// TIA Portal V16 export
// export: Created 2021-11-12T13:32:41.0114978Z, ExportSetting WithDefaults, DisplayName Totally Integrated Automation Portal, DisplayVersion V16 Update 3, DisplayName TIA Portal Version Control Interface, DisplayVersion V16 Update 2, DisplayName TIA Portal Openness, DisplayVersion V16 Update 3, DisplayName SINAMICS Startdrive Advanced, DisplayVersion V16 Update 5, DisplayName SINAMICS Startdrive G130, G150, S120, S150, SINAMICS MV, S210, DisplayVersion V16 Update 5, DisplayName SINAMICS Startdrive G110M, G120, G120C, G120D, G120P, G115D, DisplayVersion V16 Update 5, DisplayName STEP 7 Professional, DisplayVersion V16 Update 3, DisplayName STEP 7 Safety, DisplayVersion V16, DisplayName WinCC UA Professional, DisplayVersion V16 Update 3
FUNCTION_BLOCK "IM_200+UH11-KF10"   // FB26, LAD
TITLE = Inputs reading
{ S7_Optimized_Access := 'TRUE' }
VERSION : 0.1
// MICE Wood interface block
// stored: AutoNumber true, IsIECCheckEnabled false, IsRetainMemResEnabled false, MemoryReserve 100, SetENOAutomatically false, UDAEnableTagReadback false
   VAR
      KF11_Ix0 { S7_SetPoint := 'True'} : "STD_CH_DI";
      KF11_Ix1 { S7_SetPoint := 'True'} : "STD_CH_DI";
      KF11_Ix2 { S7_SetPoint := 'True'} : "STD_CH_DI";
      KF11_Ix3 { S7_SetPoint := 'True'} : "STD_CH_DI";
      KF11_Ix4 { S7_SetPoint := 'True'} : "STD_CH_DI";
      KF11_Ix5 { S7_SetPoint := 'True'} : "STD_CH_DI";
      KF11_Ix6 { S7_SetPoint := 'True'} : "STD_CH_DI";
      KF11_Ix7 { S7_SetPoint := 'True'} : "STD_CH_DI";
      KF11_Ix8 { S7_SetPoint := 'True'} : "STD_CH_DI";
      KF11_Ix9 { S7_SetPoint := 'True'} : "STD_CH_DI";
      KF11_Ix10 { S7_SetPoint := 'True'} : "STD_CH_DI";
      KF11_Ix11 { S7_SetPoint := 'True'} : "STD_CH_DI";
      KF11_Ix12 { S7_SetPoint := 'True'} : "STD_CH_DI";
      KF11_Ix13 { S7_SetPoint := 'True'} : "STD_CH_DI";
      KF11_Ix14 { S7_SetPoint := 'True'} : "STD_CH_DI";
      KF11_Ix15 { S7_SetPoint := 'True'} : "STD_CH_DI";
      KF12_Ix0 { S7_SetPoint := 'True'} : "STD_CH_DI";
      KF12_Ix1 { S7_SetPoint := 'True'} : "STD_CH_DI";
      KF12_Ix2 { S7_SetPoint := 'True'} : "STD_CH_DI";
      KF12_Ix3 { S7_SetPoint := 'True'} : "STD_CH_DI";
      KF12_Ix4 { S7_SetPoint := 'True'} : "STD_CH_DI";
      KF12_Ix5 { S7_SetPoint := 'True'} : "STD_CH_DI";
      KF12_Ix6 { S7_SetPoint := 'True'} : "STD_CH_DI";
      KF12_Ix7 { S7_SetPoint := 'True'} : "STD_CH_DI";
      KF12_Ix8 { S7_SetPoint := 'True'} : "STD_CH_DI";
      KF12_Ix9 { S7_SetPoint := 'True'} : "STD_CH_DI";
      KF12_Ix10 { S7_SetPoint := 'True'} : "STD_CH_DI";
      KF12_Ix11 { S7_SetPoint := 'True'} : "STD_CH_DI";
      KF12_Ix12 { S7_SetPoint := 'True'} : "STD_CH_DI";
      KF12_Ix13 { S7_SetPoint := 'True'} : "STD_CH_DI";
      KF12_Ix14 { S7_SetPoint := 'True'} : "STD_CH_DI";
      KF12_Ix15 { S7_SetPoint := 'True'} : "STD_CH_DI";
      KF13_Ix0 { S7_SetPoint := 'True'} : "STD_CH_DI";
      KF13_Ix1 { S7_SetPoint := 'True'} : "STD_CH_DI";
      KF13_Ix2 { S7_SetPoint := 'True'} : "STD_CH_DI";
      KF13_Ix3 { S7_SetPoint := 'True'} : "STD_CH_DI";
      KF13_Ix4 { S7_SetPoint := 'True'} : "STD_CH_DI";
      KF13_Ix5 { S7_SetPoint := 'True'} : "STD_CH_DI";
      KF13_Ix6 { S7_SetPoint := 'True'} : "STD_CH_DI";
      KF13_Ix7 { S7_SetPoint := 'True'} : "STD_CH_DI";
      KF13_Ix8 { S7_SetPoint := 'True'} : "STD_CH_DI";
      KF13_Ix9 { S7_SetPoint := 'True'} : "STD_CH_DI";
      KF13_Ix10 { S7_SetPoint := 'True'} : "STD_CH_DI";
      KF13_Ix11 { S7_SetPoint := 'True'} : "STD_CH_DI";
      KF13_Ix12 { S7_SetPoint := 'True'} : "STD_CH_DI";
      KF13_Ix13 { S7_SetPoint := 'True'} : "STD_CH_DI";
      KF13_Ix14 { S7_SetPoint := 'True'} : "STD_CH_DI";
      KF13_Ix15 { S7_SetPoint := 'True'} : "STD_CH_DI";
      KF14_Ix0 { S7_SetPoint := 'True'} : "STD_CH_DI";
      KF14_Ix1 { S7_SetPoint := 'True'} : "STD_CH_DI";
      KF14_Ix2 { S7_SetPoint := 'True'} : "STD_CH_DI";
      KF14_Ix3 { S7_SetPoint := 'True'} : "STD_CH_DI";
      KF14_Ix4 { S7_SetPoint := 'True'} : "STD_CH_DI";
      KF14_Ix5 { S7_SetPoint := 'True'} : "STD_CH_DI";
      KF14_Ix6 { S7_SetPoint := 'True'} : "STD_CH_DI";
      KF14_Ix7 { S7_SetPoint := 'True'} : "STD_CH_DI";
      KF14_Ix8 { S7_SetPoint := 'True'} : "STD_CH_DI";
      KF14_Ix9 { S7_SetPoint := 'True'} : "STD_CH_DI";
      KF14_Ix10 { S7_SetPoint := 'True'} : "STD_CH_DI";
      KF14_Ix11 { S7_SetPoint := 'True'} : "STD_CH_DI";
      KF14_Ix12 { S7_SetPoint := 'True'} : "STD_CH_DI";
      KF14_Ix13 { S7_SetPoint := 'True'} : "STD_CH_DI";
      KF14_Ix14 { S7_SetPoint := 'True'} : "STD_CH_DI";
      KF14_Ix15 { S7_SetPoint := 'True'} : "STD_CH_DI";
      KF15_Ix0 { S7_SetPoint := 'True'} : "STD_CH_DI";
      KF15_Ix1 { S7_SetPoint := 'True'} : "STD_CH_DI";
      KF15_Ix2 { S7_SetPoint := 'True'} : "STD_CH_DI";
      KF15_Ix3 { S7_SetPoint := 'True'} : "STD_CH_DI";
      KF15_Ix4 { S7_SetPoint := 'True'} : "STD_CH_DI";
      KF15_Ix5 { S7_SetPoint := 'True'} : "STD_CH_DI";
      KF15_Ix6 { S7_SetPoint := 'True'} : "STD_CH_DI";
      KF15_Ix7 { S7_SetPoint := 'True'} : "STD_CH_DI";
      KF61_AI0 { S7_SetPoint := 'True'} : "STD_CH_AI";
      KF61_AI1 { S7_SetPoint := 'True'} : "STD_CH_AI";
      KF61_AI2 { S7_SetPoint := 'True'} : "STD_CH_AI";
      KF61_AI3 { S7_SetPoint := 'True'} : "STD_CH_AI";
   END_VAR
   VAR_TEMP   // added for the SCL form of the ladder/FBD networks
      _w1 : Bool;
      _w2 : Bool;
      _w3 : Bool;
      _w4 : Bool;
      _w5 : Bool;
      _w6 : Bool;
      _w7 : Bool;
      _w8 : Bool;
   END_VAR
BEGIN

REGION Network 1: Module position -KF11
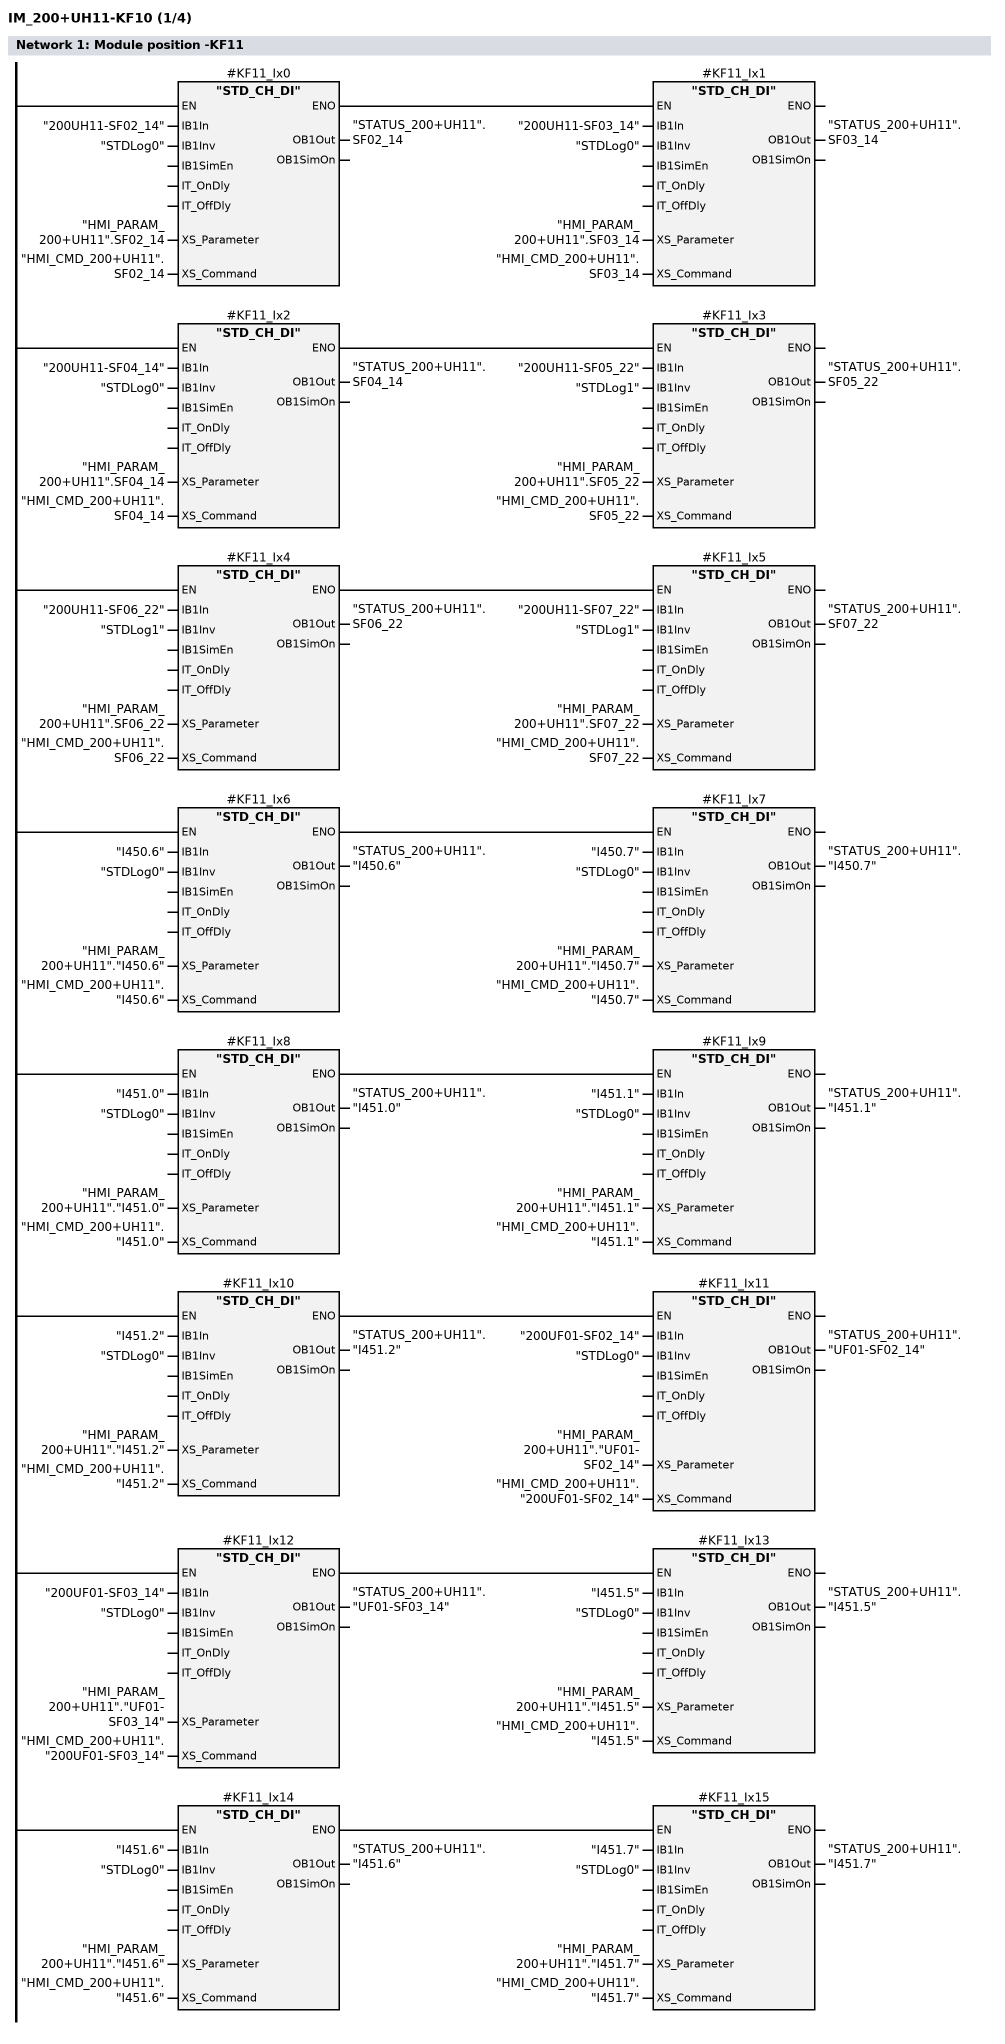
   RUNG wire#powerrail
      #KF11_Ix0(IB1In := "200UH11-SF02_14", IB1Inv := "STDLog0", IB1SimEn :=, IT_OnDly :=, IT_OffDly :=, XS_Parameter := "HMI_PARAM_200+UH11".SF02_14, XS_Command := "HMI_CMD_200+UH11".SF02_14, OB1Out => "STATUS_200+UH11".SF02_14, OB1SimOn =>)
      #KF11_Ix1(IB1In := "200UH11-SF03_14", IB1Inv := "STDLog0", IB1SimEn :=, IT_OnDly :=, IT_OffDly :=, XS_Parameter := "HMI_PARAM_200+UH11".SF03_14, XS_Command := "HMI_CMD_200+UH11".SF03_14, OB1Out => "STATUS_200+UH11".SF03_14, OB1SimOn =>)
   END_RUNG
   RUNG wire#powerrail
      #KF11_Ix2(IB1In := "200UH11-SF04_14", IB1Inv := "STDLog0", IB1SimEn :=, IT_OnDly :=, IT_OffDly :=, XS_Parameter := "HMI_PARAM_200+UH11".SF04_14, XS_Command := "HMI_CMD_200+UH11".SF04_14, OB1Out => "STATUS_200+UH11".SF04_14, OB1SimOn =>)
      #KF11_Ix3(IB1In := "200UH11-SF05_22", IB1Inv := "STDLog1", IB1SimEn :=, IT_OnDly :=, IT_OffDly :=, XS_Parameter := "HMI_PARAM_200+UH11".SF05_22, XS_Command := "HMI_CMD_200+UH11".SF05_22, OB1Out => "STATUS_200+UH11".SF05_22, OB1SimOn =>)
   END_RUNG
   RUNG wire#powerrail
      #KF11_Ix4(IB1In := "200UH11-SF06_22", IB1Inv := "STDLog1", IB1SimEn :=, IT_OnDly :=, IT_OffDly :=, XS_Parameter := "HMI_PARAM_200+UH11".SF06_22, XS_Command := "HMI_CMD_200+UH11".SF06_22, OB1Out => "STATUS_200+UH11".SF06_22, OB1SimOn =>)
      #KF11_Ix5(IB1In := "200UH11-SF07_22", IB1Inv := "STDLog1", IB1SimEn :=, IT_OnDly :=, IT_OffDly :=, XS_Parameter := "HMI_PARAM_200+UH11".SF07_22, XS_Command := "HMI_CMD_200+UH11".SF07_22, OB1Out => "STATUS_200+UH11".SF07_22, OB1SimOn =>)
   END_RUNG
   RUNG wire#powerrail
      #KF11_Ix6(IB1In := "I450.6", IB1Inv := "STDLog0", IB1SimEn :=, IT_OnDly :=, IT_OffDly :=, XS_Parameter := "HMI_PARAM_200+UH11"."I450.6", XS_Command := "HMI_CMD_200+UH11"."I450.6", OB1Out => "STATUS_200+UH11"."I450.6", OB1SimOn =>)
      #KF11_Ix7(IB1In := "I450.7", IB1Inv := "STDLog0", IB1SimEn :=, IT_OnDly :=, IT_OffDly :=, XS_Parameter := "HMI_PARAM_200+UH11"."I450.7", XS_Command := "HMI_CMD_200+UH11"."I450.7", OB1Out => "STATUS_200+UH11"."I450.7", OB1SimOn =>)
   END_RUNG
   RUNG wire#powerrail
      #KF11_Ix8(IB1In := "I451.0", IB1Inv := "STDLog0", IB1SimEn :=, IT_OnDly :=, IT_OffDly :=, XS_Parameter := "HMI_PARAM_200+UH11"."I451.0", XS_Command := "HMI_CMD_200+UH11"."I451.0", OB1Out => "STATUS_200+UH11"."I451.0", OB1SimOn =>)
      #KF11_Ix9(IB1In := "I451.1", IB1Inv := "STDLog0", IB1SimEn :=, IT_OnDly :=, IT_OffDly :=, XS_Parameter := "HMI_PARAM_200+UH11"."I451.1", XS_Command := "HMI_CMD_200+UH11"."I451.1", OB1Out => "STATUS_200+UH11"."I451.1", OB1SimOn =>)
   END_RUNG
   RUNG wire#powerrail
      #KF11_Ix10(IB1In := "I451.2", IB1Inv := "STDLog0", IB1SimEn :=, IT_OnDly :=, IT_OffDly :=, XS_Parameter := "HMI_PARAM_200+UH11"."I451.2", XS_Command := "HMI_CMD_200+UH11"."I451.2", OB1Out => "STATUS_200+UH11"."I451.2", OB1SimOn =>)
      #KF11_Ix11(IB1In := "200UF01-SF02_14", IB1Inv := "STDLog0", IB1SimEn :=, IT_OnDly :=, IT_OffDly :=, XS_Parameter := "HMI_PARAM_200+UH11"."UF01-SF02_14", XS_Command := "HMI_CMD_200+UH11"."200UF01-SF02_14", OB1Out => "STATUS_200+UH11"."UF01-SF02_14", OB1SimOn =>)
   END_RUNG
   RUNG wire#powerrail
      #KF11_Ix12(IB1In := "200UF01-SF03_14", IB1Inv := "STDLog0", IB1SimEn :=, IT_OnDly :=, IT_OffDly :=, XS_Parameter := "HMI_PARAM_200+UH11"."UF01-SF03_14", XS_Command := "HMI_CMD_200+UH11"."200UF01-SF03_14", OB1Out => "STATUS_200+UH11"."UF01-SF03_14", OB1SimOn =>)
      #KF11_Ix13(IB1In := "I451.5", IB1Inv := "STDLog0", IB1SimEn :=, IT_OnDly :=, IT_OffDly :=, XS_Parameter := "HMI_PARAM_200+UH11"."I451.5", XS_Command := "HMI_CMD_200+UH11"."I451.5", OB1Out => "STATUS_200+UH11"."I451.5", OB1SimOn =>)
   END_RUNG
   RUNG wire#powerrail
      #KF11_Ix14(IB1In := "I451.6", IB1Inv := "STDLog0", IB1SimEn :=, IT_OnDly :=, IT_OffDly :=, XS_Parameter := "HMI_PARAM_200+UH11"."I451.6", XS_Command := "HMI_CMD_200+UH11"."I451.6", OB1Out => "STATUS_200+UH11"."I451.6", OB1SimOn =>)
      #KF11_Ix15(IB1In := "I451.7", IB1Inv := "STDLog0", IB1SimEn :=, IT_OnDly :=, IT_OffDly :=, XS_Parameter := "HMI_PARAM_200+UH11"."I451.7", XS_Command := "HMI_CMD_200+UH11"."I451.7", OB1Out => "STATUS_200+UH11"."I451.7", OB1SimOn =>)
   END_RUNG
   // the same network as SCL:
   #KF11_Ix0(IB1In := "200UH11-SF02_14",   // "STD_CH_DI"
             IB1Inv := "STDLog0",
             XS_Parameter := "HMI_PARAM_200+UH11".SF02_14,
             XS_Command := "HMI_CMD_200+UH11".SF02_14,
             OB1Out => "STATUS_200+UH11".SF02_14,
             ENO => #_w1);
   IF #_w1 THEN
       #KF11_Ix1(IB1In := "200UH11-SF03_14",   // "STD_CH_DI"
                 IB1Inv := "STDLog0",
                 XS_Parameter := "HMI_PARAM_200+UH11".SF03_14,
                 XS_Command := "HMI_CMD_200+UH11".SF03_14,
                 OB1Out => "STATUS_200+UH11".SF03_14);
   END_IF;
   #KF11_Ix2(IB1In := "200UH11-SF04_14",   // "STD_CH_DI"
             IB1Inv := "STDLog0",
             XS_Parameter := "HMI_PARAM_200+UH11".SF04_14,
             XS_Command := "HMI_CMD_200+UH11".SF04_14,
             OB1Out => "STATUS_200+UH11".SF04_14,
             ENO => #_w2);
   IF #_w2 THEN
       #KF11_Ix3(IB1In := "200UH11-SF05_22",   // "STD_CH_DI"
                 IB1Inv := "STDLog1",
                 XS_Parameter := "HMI_PARAM_200+UH11".SF05_22,
                 XS_Command := "HMI_CMD_200+UH11".SF05_22,
                 OB1Out => "STATUS_200+UH11".SF05_22);
   END_IF;
   #KF11_Ix4(IB1In := "200UH11-SF06_22",   // "STD_CH_DI"
             IB1Inv := "STDLog1",
             XS_Parameter := "HMI_PARAM_200+UH11".SF06_22,
             XS_Command := "HMI_CMD_200+UH11".SF06_22,
             OB1Out => "STATUS_200+UH11".SF06_22,
             ENO => #_w3);
   IF #_w3 THEN
       #KF11_Ix5(IB1In := "200UH11-SF07_22",   // "STD_CH_DI"
                 IB1Inv := "STDLog1",
                 XS_Parameter := "HMI_PARAM_200+UH11".SF07_22,
                 XS_Command := "HMI_CMD_200+UH11".SF07_22,
                 OB1Out => "STATUS_200+UH11".SF07_22);
   END_IF;
   #KF11_Ix6(IB1In := "I450.6",   // "STD_CH_DI"
             IB1Inv := "STDLog0",
             XS_Parameter := "HMI_PARAM_200+UH11"."I450.6",
             XS_Command := "HMI_CMD_200+UH11"."I450.6",
             OB1Out => "STATUS_200+UH11"."I450.6",
             ENO => #_w4);
   IF #_w4 THEN
       #KF11_Ix7(IB1In := "I450.7",   // "STD_CH_DI"
                 IB1Inv := "STDLog0",
                 XS_Parameter := "HMI_PARAM_200+UH11"."I450.7",
                 XS_Command := "HMI_CMD_200+UH11"."I450.7",
                 OB1Out => "STATUS_200+UH11"."I450.7");
   END_IF;
   #KF11_Ix8(IB1In := "I451.0",   // "STD_CH_DI"
             IB1Inv := "STDLog0",
             XS_Parameter := "HMI_PARAM_200+UH11"."I451.0",
             XS_Command := "HMI_CMD_200+UH11"."I451.0",
             OB1Out => "STATUS_200+UH11"."I451.0",
             ENO => #_w5);
   IF #_w5 THEN
       #KF11_Ix9(IB1In := "I451.1",   // "STD_CH_DI"
                 IB1Inv := "STDLog0",
                 XS_Parameter := "HMI_PARAM_200+UH11"."I451.1",
                 XS_Command := "HMI_CMD_200+UH11"."I451.1",
                 OB1Out => "STATUS_200+UH11"."I451.1");
   END_IF;
   #KF11_Ix10(IB1In := "I451.2",   // "STD_CH_DI"
              IB1Inv := "STDLog0",
              XS_Parameter := "HMI_PARAM_200+UH11"."I451.2",
              XS_Command := "HMI_CMD_200+UH11"."I451.2",
              OB1Out => "STATUS_200+UH11"."I451.2",
              ENO => #_w6);
   IF #_w6 THEN
       #KF11_Ix11(IB1In := "200UF01-SF02_14",   // "STD_CH_DI"
                  IB1Inv := "STDLog0",
                  XS_Parameter := "HMI_PARAM_200+UH11"."UF01-SF02_14",
                  XS_Command := "HMI_CMD_200+UH11"."200UF01-SF02_14",
                  OB1Out => "STATUS_200+UH11"."UF01-SF02_14");
   END_IF;
   #KF11_Ix12(IB1In := "200UF01-SF03_14",   // "STD_CH_DI"
              IB1Inv := "STDLog0",
              XS_Parameter := "HMI_PARAM_200+UH11"."UF01-SF03_14",
              XS_Command := "HMI_CMD_200+UH11"."200UF01-SF03_14",
              OB1Out => "STATUS_200+UH11"."UF01-SF03_14",
              ENO => #_w7);
   IF #_w7 THEN
       #KF11_Ix13(IB1In := "I451.5",   // "STD_CH_DI"
                  IB1Inv := "STDLog0",
                  XS_Parameter := "HMI_PARAM_200+UH11"."I451.5",
                  XS_Command := "HMI_CMD_200+UH11"."I451.5",
                  OB1Out => "STATUS_200+UH11"."I451.5");
   END_IF;
   #KF11_Ix14(IB1In := "I451.6",   // "STD_CH_DI"
              IB1Inv := "STDLog0",
              XS_Parameter := "HMI_PARAM_200+UH11"."I451.6",
              XS_Command := "HMI_CMD_200+UH11"."I451.6",
              OB1Out => "STATUS_200+UH11"."I451.6",
              ENO => #_w8);
   IF #_w8 THEN
       #KF11_Ix15(IB1In := "I451.7",   // "STD_CH_DI"
                  IB1Inv := "STDLog0",
                  XS_Parameter := "HMI_PARAM_200+UH11"."I451.7",
                  XS_Command := "HMI_CMD_200+UH11"."I451.7",
                  OB1Out => "STATUS_200+UH11"."I451.7");
   END_IF;
END_REGION

REGION Network 2: Module position -KF12
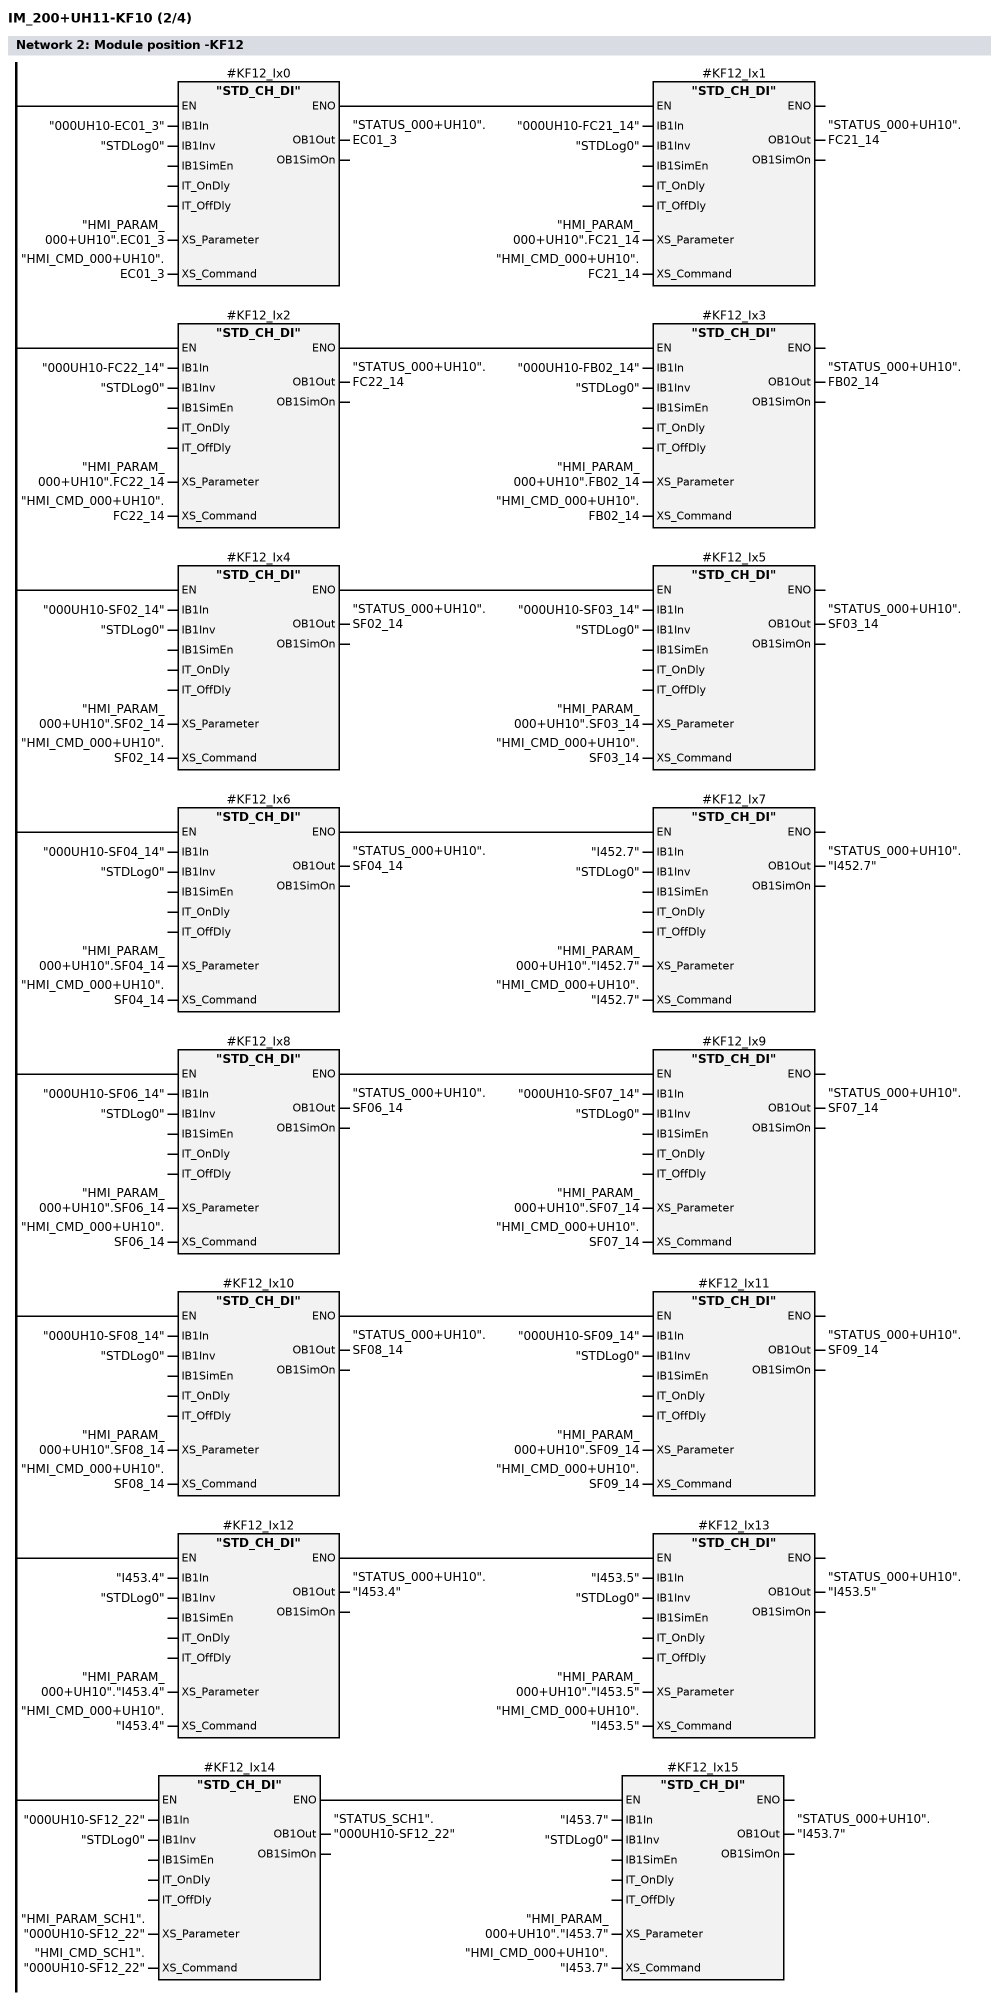
   RUNG wire#powerrail
      #KF12_Ix0(IB1In := "000UH10-EC01_3", IB1Inv := "STDLog0", IB1SimEn :=, IT_OnDly :=, IT_OffDly :=, XS_Parameter := "HMI_PARAM_000+UH10".EC01_3, XS_Command := "HMI_CMD_000+UH10".EC01_3, OB1Out => "STATUS_000+UH10".EC01_3, OB1SimOn =>)
      #KF12_Ix1(IB1In := "000UH10-FC21_14", IB1Inv := "STDLog0", IB1SimEn :=, IT_OnDly :=, IT_OffDly :=, XS_Parameter := "HMI_PARAM_000+UH10".FC21_14, XS_Command := "HMI_CMD_000+UH10".FC21_14, OB1Out => "STATUS_000+UH10".FC21_14, OB1SimOn =>)
   END_RUNG
   RUNG wire#powerrail
      #KF12_Ix2(IB1In := "000UH10-FC22_14", IB1Inv := "STDLog0", IB1SimEn :=, IT_OnDly :=, IT_OffDly :=, XS_Parameter := "HMI_PARAM_000+UH10".FC22_14, XS_Command := "HMI_CMD_000+UH10".FC22_14, OB1Out => "STATUS_000+UH10".FC22_14, OB1SimOn =>)
      #KF12_Ix3(IB1In := "000UH10-FB02_14", IB1Inv := "STDLog0", IB1SimEn :=, IT_OnDly :=, IT_OffDly :=, XS_Parameter := "HMI_PARAM_000+UH10".FB02_14, XS_Command := "HMI_CMD_000+UH10".FB02_14, OB1Out => "STATUS_000+UH10".FB02_14, OB1SimOn =>)
   END_RUNG
   RUNG wire#powerrail
      #KF12_Ix4(IB1In := "000UH10-SF02_14", IB1Inv := "STDLog0", IB1SimEn :=, IT_OnDly :=, IT_OffDly :=, XS_Parameter := "HMI_PARAM_000+UH10".SF02_14, XS_Command := "HMI_CMD_000+UH10".SF02_14, OB1Out => "STATUS_000+UH10".SF02_14, OB1SimOn =>)
      #KF12_Ix5(IB1In := "000UH10-SF03_14", IB1Inv := "STDLog0", IB1SimEn :=, IT_OnDly :=, IT_OffDly :=, XS_Parameter := "HMI_PARAM_000+UH10".SF03_14, XS_Command := "HMI_CMD_000+UH10".SF03_14, OB1Out => "STATUS_000+UH10".SF03_14, OB1SimOn =>)
   END_RUNG
   RUNG wire#powerrail
      #KF12_Ix6(IB1In := "000UH10-SF04_14", IB1Inv := "STDLog0", IB1SimEn :=, IT_OnDly :=, IT_OffDly :=, XS_Parameter := "HMI_PARAM_000+UH10".SF04_14, XS_Command := "HMI_CMD_000+UH10".SF04_14, OB1Out => "STATUS_000+UH10".SF04_14, OB1SimOn =>)
      #KF12_Ix7(IB1In := "I452.7", IB1Inv := "STDLog0", IB1SimEn :=, IT_OnDly :=, IT_OffDly :=, XS_Parameter := "HMI_PARAM_000+UH10"."I452.7", XS_Command := "HMI_CMD_000+UH10"."I452.7", OB1Out => "STATUS_000+UH10"."I452.7", OB1SimOn =>)
   END_RUNG
   RUNG wire#powerrail
      #KF12_Ix8(IB1In := "000UH10-SF06_14", IB1Inv := "STDLog0", IB1SimEn :=, IT_OnDly :=, IT_OffDly :=, XS_Parameter := "HMI_PARAM_000+UH10".SF06_14, XS_Command := "HMI_CMD_000+UH10".SF06_14, OB1Out => "STATUS_000+UH10".SF06_14, OB1SimOn =>)
      #KF12_Ix9(IB1In := "000UH10-SF07_14", IB1Inv := "STDLog0", IB1SimEn :=, IT_OnDly :=, IT_OffDly :=, XS_Parameter := "HMI_PARAM_000+UH10".SF07_14, XS_Command := "HMI_CMD_000+UH10".SF07_14, OB1Out => "STATUS_000+UH10".SF07_14, OB1SimOn =>)
   END_RUNG
   RUNG wire#powerrail
      #KF12_Ix10(IB1In := "000UH10-SF08_14", IB1Inv := "STDLog0", IB1SimEn :=, IT_OnDly :=, IT_OffDly :=, XS_Parameter := "HMI_PARAM_000+UH10".SF08_14, XS_Command := "HMI_CMD_000+UH10".SF08_14, OB1Out => "STATUS_000+UH10".SF08_14, OB1SimOn =>)
      #KF12_Ix11(IB1In := "000UH10-SF09_14", IB1Inv := "STDLog0", IB1SimEn :=, IT_OnDly :=, IT_OffDly :=, XS_Parameter := "HMI_PARAM_000+UH10".SF09_14, XS_Command := "HMI_CMD_000+UH10".SF09_14, OB1Out => "STATUS_000+UH10".SF09_14, OB1SimOn =>)
   END_RUNG
   RUNG wire#powerrail
      #KF12_Ix12(IB1In := "I453.4", IB1Inv := "STDLog0", IB1SimEn :=, IT_OnDly :=, IT_OffDly :=, XS_Parameter := "HMI_PARAM_000+UH10"."I453.4", XS_Command := "HMI_CMD_000+UH10"."I453.4", OB1Out => "STATUS_000+UH10"."I453.4", OB1SimOn =>)
      #KF12_Ix13(IB1In := "I453.5", IB1Inv := "STDLog0", IB1SimEn :=, IT_OnDly :=, IT_OffDly :=, XS_Parameter := "HMI_PARAM_000+UH10"."I453.5", XS_Command := "HMI_CMD_000+UH10"."I453.5", OB1Out => "STATUS_000+UH10"."I453.5", OB1SimOn =>)
   END_RUNG
   RUNG wire#powerrail
      #KF12_Ix14(IB1In := "000UH10-SF12_22", IB1Inv := "STDLog0", IB1SimEn :=, IT_OnDly :=, IT_OffDly :=, XS_Parameter := "HMI_PARAM_SCH1"."000UH10-SF12_22", XS_Command := "HMI_CMD_SCH1"."000UH10-SF12_22", OB1Out => "STATUS_SCH1"."000UH10-SF12_22", OB1SimOn =>)
      #KF12_Ix15(IB1In := "I453.7", IB1Inv := "STDLog0", IB1SimEn :=, IT_OnDly :=, IT_OffDly :=, XS_Parameter := "HMI_PARAM_000+UH10"."I453.7", XS_Command := "HMI_CMD_000+UH10"."I453.7", OB1Out => "STATUS_000+UH10"."I453.7", OB1SimOn =>)
   END_RUNG
   // the same network as SCL:
   #KF12_Ix0(IB1In := "000UH10-EC01_3",   // "STD_CH_DI"
             IB1Inv := "STDLog0",
             XS_Parameter := "HMI_PARAM_000+UH10".EC01_3,
             XS_Command := "HMI_CMD_000+UH10".EC01_3,
             OB1Out => "STATUS_000+UH10".EC01_3,
             ENO => #_w1);
   IF #_w1 THEN
       #KF12_Ix1(IB1In := "000UH10-FC21_14",   // "STD_CH_DI"
                 IB1Inv := "STDLog0",
                 XS_Parameter := "HMI_PARAM_000+UH10".FC21_14,
                 XS_Command := "HMI_CMD_000+UH10".FC21_14,
                 OB1Out => "STATUS_000+UH10".FC21_14);
   END_IF;
   #KF12_Ix2(IB1In := "000UH10-FC22_14",   // "STD_CH_DI"
             IB1Inv := "STDLog0",
             XS_Parameter := "HMI_PARAM_000+UH10".FC22_14,
             XS_Command := "HMI_CMD_000+UH10".FC22_14,
             OB1Out => "STATUS_000+UH10".FC22_14,
             ENO => #_w2);
   IF #_w2 THEN
       #KF12_Ix3(IB1In := "000UH10-FB02_14",   // "STD_CH_DI"
                 IB1Inv := "STDLog0",
                 XS_Parameter := "HMI_PARAM_000+UH10".FB02_14,
                 XS_Command := "HMI_CMD_000+UH10".FB02_14,
                 OB1Out => "STATUS_000+UH10".FB02_14);
   END_IF;
   #KF12_Ix4(IB1In := "000UH10-SF02_14",   // "STD_CH_DI"
             IB1Inv := "STDLog0",
             XS_Parameter := "HMI_PARAM_000+UH10".SF02_14,
             XS_Command := "HMI_CMD_000+UH10".SF02_14,
             OB1Out => "STATUS_000+UH10".SF02_14,
             ENO => #_w3);
   IF #_w3 THEN
       #KF12_Ix5(IB1In := "000UH10-SF03_14",   // "STD_CH_DI"
                 IB1Inv := "STDLog0",
                 XS_Parameter := "HMI_PARAM_000+UH10".SF03_14,
                 XS_Command := "HMI_CMD_000+UH10".SF03_14,
                 OB1Out => "STATUS_000+UH10".SF03_14);
   END_IF;
   #KF12_Ix6(IB1In := "000UH10-SF04_14",   // "STD_CH_DI"
             IB1Inv := "STDLog0",
             XS_Parameter := "HMI_PARAM_000+UH10".SF04_14,
             XS_Command := "HMI_CMD_000+UH10".SF04_14,
             OB1Out => "STATUS_000+UH10".SF04_14,
             ENO => #_w4);
   IF #_w4 THEN
       #KF12_Ix7(IB1In := "I452.7",   // "STD_CH_DI"
                 IB1Inv := "STDLog0",
                 XS_Parameter := "HMI_PARAM_000+UH10"."I452.7",
                 XS_Command := "HMI_CMD_000+UH10"."I452.7",
                 OB1Out => "STATUS_000+UH10"."I452.7");
   END_IF;
   #KF12_Ix8(IB1In := "000UH10-SF06_14",   // "STD_CH_DI"
             IB1Inv := "STDLog0",
             XS_Parameter := "HMI_PARAM_000+UH10".SF06_14,
             XS_Command := "HMI_CMD_000+UH10".SF06_14,
             OB1Out => "STATUS_000+UH10".SF06_14,
             ENO => #_w5);
   IF #_w5 THEN
       #KF12_Ix9(IB1In := "000UH10-SF07_14",   // "STD_CH_DI"
                 IB1Inv := "STDLog0",
                 XS_Parameter := "HMI_PARAM_000+UH10".SF07_14,
                 XS_Command := "HMI_CMD_000+UH10".SF07_14,
                 OB1Out => "STATUS_000+UH10".SF07_14);
   END_IF;
   #KF12_Ix10(IB1In := "000UH10-SF08_14",   // "STD_CH_DI"
              IB1Inv := "STDLog0",
              XS_Parameter := "HMI_PARAM_000+UH10".SF08_14,
              XS_Command := "HMI_CMD_000+UH10".SF08_14,
              OB1Out => "STATUS_000+UH10".SF08_14,
              ENO => #_w6);
   IF #_w6 THEN
       #KF12_Ix11(IB1In := "000UH10-SF09_14",   // "STD_CH_DI"
                  IB1Inv := "STDLog0",
                  XS_Parameter := "HMI_PARAM_000+UH10".SF09_14,
                  XS_Command := "HMI_CMD_000+UH10".SF09_14,
                  OB1Out => "STATUS_000+UH10".SF09_14);
   END_IF;
   #KF12_Ix12(IB1In := "I453.4",   // "STD_CH_DI"
              IB1Inv := "STDLog0",
              XS_Parameter := "HMI_PARAM_000+UH10"."I453.4",
              XS_Command := "HMI_CMD_000+UH10"."I453.4",
              OB1Out => "STATUS_000+UH10"."I453.4",
              ENO => #_w7);
   IF #_w7 THEN
       #KF12_Ix13(IB1In := "I453.5",   // "STD_CH_DI"
                  IB1Inv := "STDLog0",
                  XS_Parameter := "HMI_PARAM_000+UH10"."I453.5",
                  XS_Command := "HMI_CMD_000+UH10"."I453.5",
                  OB1Out => "STATUS_000+UH10"."I453.5");
   END_IF;
   #KF12_Ix14(IB1In := "000UH10-SF12_22",   // "STD_CH_DI"
              IB1Inv := "STDLog0",
              XS_Parameter := "HMI_PARAM_SCH1"."000UH10-SF12_22",
              XS_Command := "HMI_CMD_SCH1"."000UH10-SF12_22",
              OB1Out => "STATUS_SCH1"."000UH10-SF12_22",
              ENO => #_w8);
   IF #_w8 THEN
       #KF12_Ix15(IB1In := "I453.7",   // "STD_CH_DI"
                  IB1Inv := "STDLog0",
                  XS_Parameter := "HMI_PARAM_000+UH10"."I453.7",
                  XS_Command := "HMI_CMD_000+UH10"."I453.7",
                  OB1Out => "STATUS_000+UH10"."I453.7");
   END_IF;
END_REGION

REGION Network 3: Module position -KF13
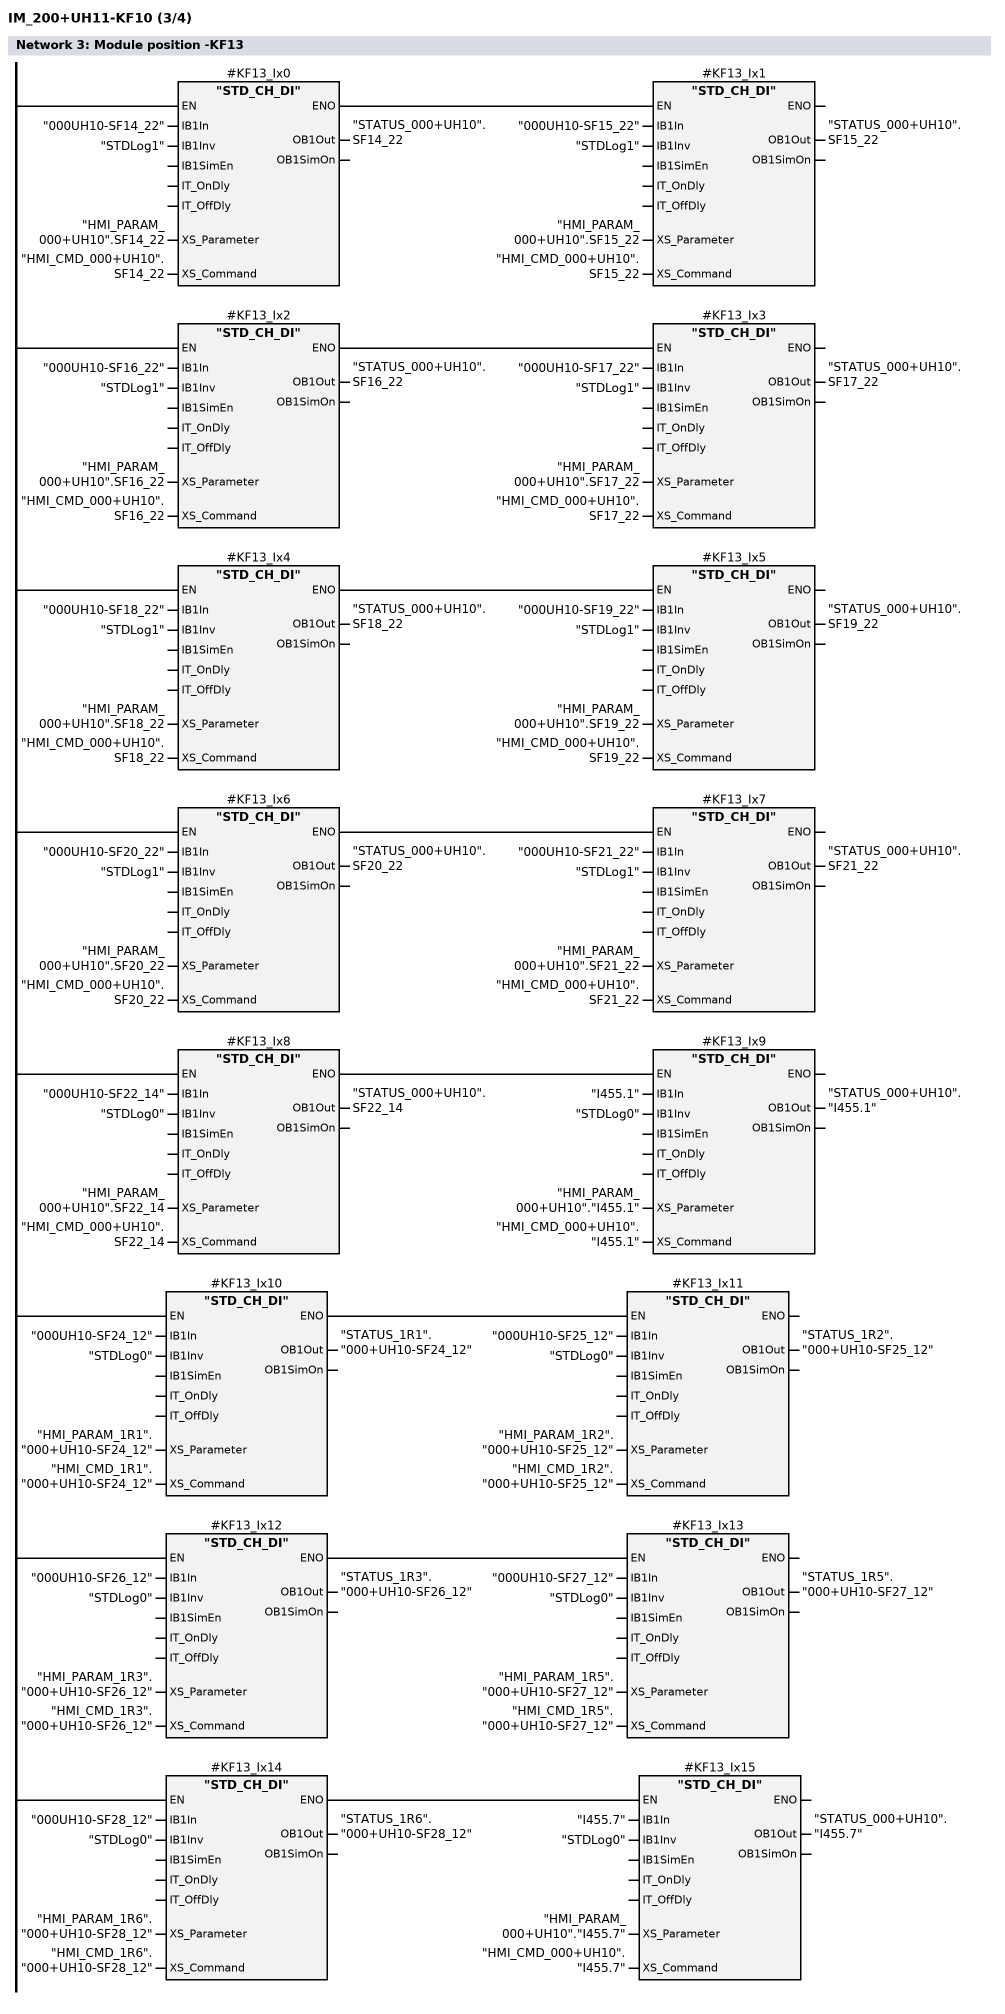
   RUNG wire#powerrail
      #KF13_Ix0(IB1In := "000UH10-SF14_22", IB1Inv := "STDLog1", IB1SimEn :=, IT_OnDly :=, IT_OffDly :=, XS_Parameter := "HMI_PARAM_000+UH10".SF14_22, XS_Command := "HMI_CMD_000+UH10".SF14_22, OB1Out => "STATUS_000+UH10".SF14_22, OB1SimOn =>)
      #KF13_Ix1(IB1In := "000UH10-SF15_22", IB1Inv := "STDLog1", IB1SimEn :=, IT_OnDly :=, IT_OffDly :=, XS_Parameter := "HMI_PARAM_000+UH10".SF15_22, XS_Command := "HMI_CMD_000+UH10".SF15_22, OB1Out => "STATUS_000+UH10".SF15_22, OB1SimOn =>)
   END_RUNG
   RUNG wire#powerrail
      #KF13_Ix2(IB1In := "000UH10-SF16_22", IB1Inv := "STDLog1", IB1SimEn :=, IT_OnDly :=, IT_OffDly :=, XS_Parameter := "HMI_PARAM_000+UH10".SF16_22, XS_Command := "HMI_CMD_000+UH10".SF16_22, OB1Out => "STATUS_000+UH10".SF16_22, OB1SimOn =>)
      #KF13_Ix3(IB1In := "000UH10-SF17_22", IB1Inv := "STDLog1", IB1SimEn :=, IT_OnDly :=, IT_OffDly :=, XS_Parameter := "HMI_PARAM_000+UH10".SF17_22, XS_Command := "HMI_CMD_000+UH10".SF17_22, OB1Out => "STATUS_000+UH10".SF17_22, OB1SimOn =>)
   END_RUNG
   RUNG wire#powerrail
      #KF13_Ix4(IB1In := "000UH10-SF18_22", IB1Inv := "STDLog1", IB1SimEn :=, IT_OnDly :=, IT_OffDly :=, XS_Parameter := "HMI_PARAM_000+UH10".SF18_22, XS_Command := "HMI_CMD_000+UH10".SF18_22, OB1Out => "STATUS_000+UH10".SF18_22, OB1SimOn =>)
      #KF13_Ix5(IB1In := "000UH10-SF19_22", IB1Inv := "STDLog1", IB1SimEn :=, IT_OnDly :=, IT_OffDly :=, XS_Parameter := "HMI_PARAM_000+UH10".SF19_22, XS_Command := "HMI_CMD_000+UH10".SF19_22, OB1Out => "STATUS_000+UH10".SF19_22, OB1SimOn =>)
   END_RUNG
   RUNG wire#powerrail
      #KF13_Ix6(IB1In := "000UH10-SF20_22", IB1Inv := "STDLog1", IB1SimEn :=, IT_OnDly :=, IT_OffDly :=, XS_Parameter := "HMI_PARAM_000+UH10".SF20_22, XS_Command := "HMI_CMD_000+UH10".SF20_22, OB1Out => "STATUS_000+UH10".SF20_22, OB1SimOn =>)
      #KF13_Ix7(IB1In := "000UH10-SF21_22", IB1Inv := "STDLog1", IB1SimEn :=, IT_OnDly :=, IT_OffDly :=, XS_Parameter := "HMI_PARAM_000+UH10".SF21_22, XS_Command := "HMI_CMD_000+UH10".SF21_22, OB1Out => "STATUS_000+UH10".SF21_22, OB1SimOn =>)
   END_RUNG
   RUNG wire#powerrail
      #KF13_Ix8(IB1In := "000UH10-SF22_14", IB1Inv := "STDLog0", IB1SimEn :=, IT_OnDly :=, IT_OffDly :=, XS_Parameter := "HMI_PARAM_000+UH10".SF22_14, XS_Command := "HMI_CMD_000+UH10".SF22_14, OB1Out => "STATUS_000+UH10".SF22_14, OB1SimOn =>)
      #KF13_Ix9(IB1In := "I455.1", IB1Inv := "STDLog0", IB1SimEn :=, IT_OnDly :=, IT_OffDly :=, XS_Parameter := "HMI_PARAM_000+UH10"."I455.1", XS_Command := "HMI_CMD_000+UH10"."I455.1", OB1Out => "STATUS_000+UH10"."I455.1", OB1SimOn =>)
   END_RUNG
   RUNG wire#powerrail
      #KF13_Ix10(IB1In := "000UH10-SF24_12", IB1Inv := "STDLog0", IB1SimEn :=, IT_OnDly :=, IT_OffDly :=, XS_Parameter := "HMI_PARAM_1R1"."000+UH10-SF24_12", XS_Command := "HMI_CMD_1R1"."000+UH10-SF24_12", OB1Out => "STATUS_1R1"."000+UH10-SF24_12", OB1SimOn =>)
      #KF13_Ix11(IB1In := "000UH10-SF25_12", IB1Inv := "STDLog0", IB1SimEn :=, IT_OnDly :=, IT_OffDly :=, XS_Parameter := "HMI_PARAM_1R2"."000+UH10-SF25_12", XS_Command := "HMI_CMD_1R2"."000+UH10-SF25_12", OB1Out => "STATUS_1R2"."000+UH10-SF25_12", OB1SimOn =>)
   END_RUNG
   RUNG wire#powerrail
      #KF13_Ix12(IB1In := "000UH10-SF26_12", IB1Inv := "STDLog0", IB1SimEn :=, IT_OnDly :=, IT_OffDly :=, XS_Parameter := "HMI_PARAM_1R3"."000+UH10-SF26_12", XS_Command := "HMI_CMD_1R3"."000+UH10-SF26_12", OB1Out => "STATUS_1R3"."000+UH10-SF26_12", OB1SimOn =>)
      #KF13_Ix13(IB1In := "000UH10-SF27_12", IB1Inv := "STDLog0", IB1SimEn :=, IT_OnDly :=, IT_OffDly :=, XS_Parameter := "HMI_PARAM_1R5"."000+UH10-SF27_12", XS_Command := "HMI_CMD_1R5"."000+UH10-SF27_12", OB1Out => "STATUS_1R5"."000+UH10-SF27_12", OB1SimOn =>)
   END_RUNG
   RUNG wire#powerrail
      #KF13_Ix14(IB1In := "000UH10-SF28_12", IB1Inv := "STDLog0", IB1SimEn :=, IT_OnDly :=, IT_OffDly :=, XS_Parameter := "HMI_PARAM_1R6"."000+UH10-SF28_12", XS_Command := "HMI_CMD_1R6"."000+UH10-SF28_12", OB1Out => "STATUS_1R6"."000+UH10-SF28_12", OB1SimOn =>)
      #KF13_Ix15(IB1In := "I455.7", IB1Inv := "STDLog0", IB1SimEn :=, IT_OnDly :=, IT_OffDly :=, XS_Parameter := "HMI_PARAM_000+UH10"."I455.7", XS_Command := "HMI_CMD_000+UH10"."I455.7", OB1Out => "STATUS_000+UH10"."I455.7", OB1SimOn =>)
   END_RUNG
   // the same network as SCL:
   #KF13_Ix0(IB1In := "000UH10-SF14_22",   // "STD_CH_DI"
             IB1Inv := "STDLog1",
             XS_Parameter := "HMI_PARAM_000+UH10".SF14_22,
             XS_Command := "HMI_CMD_000+UH10".SF14_22,
             OB1Out => "STATUS_000+UH10".SF14_22,
             ENO => #_w1);
   IF #_w1 THEN
       #KF13_Ix1(IB1In := "000UH10-SF15_22",   // "STD_CH_DI"
                 IB1Inv := "STDLog1",
                 XS_Parameter := "HMI_PARAM_000+UH10".SF15_22,
                 XS_Command := "HMI_CMD_000+UH10".SF15_22,
                 OB1Out => "STATUS_000+UH10".SF15_22);
   END_IF;
   #KF13_Ix2(IB1In := "000UH10-SF16_22",   // "STD_CH_DI"
             IB1Inv := "STDLog1",
             XS_Parameter := "HMI_PARAM_000+UH10".SF16_22,
             XS_Command := "HMI_CMD_000+UH10".SF16_22,
             OB1Out => "STATUS_000+UH10".SF16_22,
             ENO => #_w2);
   IF #_w2 THEN
       #KF13_Ix3(IB1In := "000UH10-SF17_22",   // "STD_CH_DI"
                 IB1Inv := "STDLog1",
                 XS_Parameter := "HMI_PARAM_000+UH10".SF17_22,
                 XS_Command := "HMI_CMD_000+UH10".SF17_22,
                 OB1Out => "STATUS_000+UH10".SF17_22);
   END_IF;
   #KF13_Ix4(IB1In := "000UH10-SF18_22",   // "STD_CH_DI"
             IB1Inv := "STDLog1",
             XS_Parameter := "HMI_PARAM_000+UH10".SF18_22,
             XS_Command := "HMI_CMD_000+UH10".SF18_22,
             OB1Out => "STATUS_000+UH10".SF18_22,
             ENO => #_w3);
   IF #_w3 THEN
       #KF13_Ix5(IB1In := "000UH10-SF19_22",   // "STD_CH_DI"
                 IB1Inv := "STDLog1",
                 XS_Parameter := "HMI_PARAM_000+UH10".SF19_22,
                 XS_Command := "HMI_CMD_000+UH10".SF19_22,
                 OB1Out => "STATUS_000+UH10".SF19_22);
   END_IF;
   #KF13_Ix6(IB1In := "000UH10-SF20_22",   // "STD_CH_DI"
             IB1Inv := "STDLog1",
             XS_Parameter := "HMI_PARAM_000+UH10".SF20_22,
             XS_Command := "HMI_CMD_000+UH10".SF20_22,
             OB1Out => "STATUS_000+UH10".SF20_22,
             ENO => #_w4);
   IF #_w4 THEN
       #KF13_Ix7(IB1In := "000UH10-SF21_22",   // "STD_CH_DI"
                 IB1Inv := "STDLog1",
                 XS_Parameter := "HMI_PARAM_000+UH10".SF21_22,
                 XS_Command := "HMI_CMD_000+UH10".SF21_22,
                 OB1Out => "STATUS_000+UH10".SF21_22);
   END_IF;
   #KF13_Ix8(IB1In := "000UH10-SF22_14",   // "STD_CH_DI"
             IB1Inv := "STDLog0",
             XS_Parameter := "HMI_PARAM_000+UH10".SF22_14,
             XS_Command := "HMI_CMD_000+UH10".SF22_14,
             OB1Out => "STATUS_000+UH10".SF22_14,
             ENO => #_w5);
   IF #_w5 THEN
       #KF13_Ix9(IB1In := "I455.1",   // "STD_CH_DI"
                 IB1Inv := "STDLog0",
                 XS_Parameter := "HMI_PARAM_000+UH10"."I455.1",
                 XS_Command := "HMI_CMD_000+UH10"."I455.1",
                 OB1Out => "STATUS_000+UH10"."I455.1");
   END_IF;
   #KF13_Ix10(IB1In := "000UH10-SF24_12",   // "STD_CH_DI"
              IB1Inv := "STDLog0",
              XS_Parameter := "HMI_PARAM_1R1"."000+UH10-SF24_12",
              XS_Command := "HMI_CMD_1R1"."000+UH10-SF24_12",
              OB1Out => "STATUS_1R1"."000+UH10-SF24_12",
              ENO => #_w6);
   IF #_w6 THEN
       #KF13_Ix11(IB1In := "000UH10-SF25_12",   // "STD_CH_DI"
                  IB1Inv := "STDLog0",
                  XS_Parameter := "HMI_PARAM_1R2"."000+UH10-SF25_12",
                  XS_Command := "HMI_CMD_1R2"."000+UH10-SF25_12",
                  OB1Out => "STATUS_1R2"."000+UH10-SF25_12");
   END_IF;
   #KF13_Ix12(IB1In := "000UH10-SF26_12",   // "STD_CH_DI"
              IB1Inv := "STDLog0",
              XS_Parameter := "HMI_PARAM_1R3"."000+UH10-SF26_12",
              XS_Command := "HMI_CMD_1R3"."000+UH10-SF26_12",
              OB1Out => "STATUS_1R3"."000+UH10-SF26_12",
              ENO => #_w7);
   IF #_w7 THEN
       #KF13_Ix13(IB1In := "000UH10-SF27_12",   // "STD_CH_DI"
                  IB1Inv := "STDLog0",
                  XS_Parameter := "HMI_PARAM_1R5"."000+UH10-SF27_12",
                  XS_Command := "HMI_CMD_1R5"."000+UH10-SF27_12",
                  OB1Out => "STATUS_1R5"."000+UH10-SF27_12");
   END_IF;
   #KF13_Ix14(IB1In := "000UH10-SF28_12",   // "STD_CH_DI"
              IB1Inv := "STDLog0",
              XS_Parameter := "HMI_PARAM_1R6"."000+UH10-SF28_12",
              XS_Command := "HMI_CMD_1R6"."000+UH10-SF28_12",
              OB1Out => "STATUS_1R6"."000+UH10-SF28_12",
              ENO => #_w8);
   IF #_w8 THEN
       #KF13_Ix15(IB1In := "I455.7",   // "STD_CH_DI"
                  IB1Inv := "STDLog0",
                  XS_Parameter := "HMI_PARAM_000+UH10"."I455.7",
                  XS_Command := "HMI_CMD_000+UH10"."I455.7",
                  OB1Out => "STATUS_000+UH10"."I455.7");
   END_IF;
END_REGION

REGION Network 4: Module position - KF14
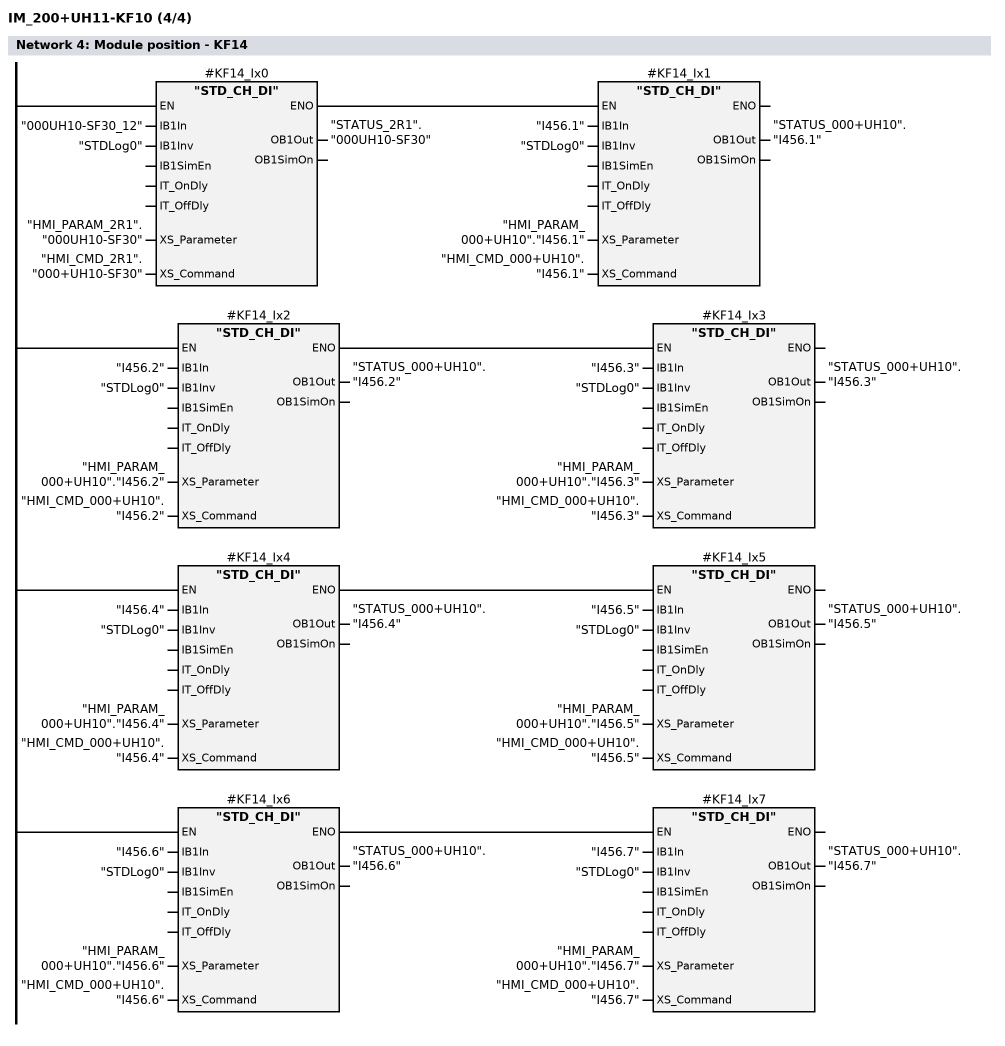
   RUNG wire#powerrail
      #KF14_Ix0(IB1In := "000UH10-SF30_12", IB1Inv := "STDLog0", IB1SimEn :=, IT_OnDly :=, IT_OffDly :=, XS_Parameter := "HMI_PARAM_2R1"."000UH10-SF30", XS_Command := "HMI_CMD_2R1"."000+UH10-SF30", OB1Out => "STATUS_2R1"."000UH10-SF30", OB1SimOn =>)
      #KF14_Ix1(IB1In := "I456.1", IB1Inv := "STDLog0", IB1SimEn :=, IT_OnDly :=, IT_OffDly :=, XS_Parameter := "HMI_PARAM_000+UH10"."I456.1", XS_Command := "HMI_CMD_000+UH10"."I456.1", OB1Out => "STATUS_000+UH10"."I456.1", OB1SimOn =>)
   END_RUNG
   RUNG wire#powerrail
      #KF14_Ix2(IB1In := "I456.2", IB1Inv := "STDLog0", IB1SimEn :=, IT_OnDly :=, IT_OffDly :=, XS_Parameter := "HMI_PARAM_000+UH10"."I456.2", XS_Command := "HMI_CMD_000+UH10"."I456.2", OB1Out => "STATUS_000+UH10"."I456.2", OB1SimOn =>)
      #KF14_Ix3(IB1In := "I456.3", IB1Inv := "STDLog0", IB1SimEn :=, IT_OnDly :=, IT_OffDly :=, XS_Parameter := "HMI_PARAM_000+UH10"."I456.3", XS_Command := "HMI_CMD_000+UH10"."I456.3", OB1Out => "STATUS_000+UH10"."I456.3", OB1SimOn =>)
   END_RUNG
   RUNG wire#powerrail
      #KF14_Ix4(IB1In := "I456.4", IB1Inv := "STDLog0", IB1SimEn :=, IT_OnDly :=, IT_OffDly :=, XS_Parameter := "HMI_PARAM_000+UH10"."I456.4", XS_Command := "HMI_CMD_000+UH10"."I456.4", OB1Out => "STATUS_000+UH10"."I456.4", OB1SimOn =>)
      #KF14_Ix5(IB1In := "I456.5", IB1Inv := "STDLog0", IB1SimEn :=, IT_OnDly :=, IT_OffDly :=, XS_Parameter := "HMI_PARAM_000+UH10"."I456.5", XS_Command := "HMI_CMD_000+UH10"."I456.5", OB1Out => "STATUS_000+UH10"."I456.5", OB1SimOn =>)
   END_RUNG
   RUNG wire#powerrail
      #KF14_Ix6(IB1In := "I456.6", IB1Inv := "STDLog0", IB1SimEn :=, IT_OnDly :=, IT_OffDly :=, XS_Parameter := "HMI_PARAM_000+UH10"."I456.6", XS_Command := "HMI_CMD_000+UH10"."I456.6", OB1Out => "STATUS_000+UH10"."I456.6", OB1SimOn =>)
      #KF14_Ix7(IB1In := "I456.7", IB1Inv := "STDLog0", IB1SimEn :=, IT_OnDly :=, IT_OffDly :=, XS_Parameter := "HMI_PARAM_000+UH10"."I456.7", XS_Command := "HMI_CMD_000+UH10"."I456.7", OB1Out => "STATUS_000+UH10"."I456.7", OB1SimOn =>)
   END_RUNG
   // the same network as SCL:
   #KF14_Ix0(IB1In := "000UH10-SF30_12",   // "STD_CH_DI"
             IB1Inv := "STDLog0",
             XS_Parameter := "HMI_PARAM_2R1"."000UH10-SF30",
             XS_Command := "HMI_CMD_2R1"."000+UH10-SF30",
             OB1Out => "STATUS_2R1"."000UH10-SF30",
             ENO => #_w1);
   IF #_w1 THEN
       #KF14_Ix1(IB1In := "I456.1",   // "STD_CH_DI"
                 IB1Inv := "STDLog0",
                 XS_Parameter := "HMI_PARAM_000+UH10"."I456.1",
                 XS_Command := "HMI_CMD_000+UH10"."I456.1",
                 OB1Out => "STATUS_000+UH10"."I456.1");
   END_IF;
   #KF14_Ix2(IB1In := "I456.2",   // "STD_CH_DI"
             IB1Inv := "STDLog0",
             XS_Parameter := "HMI_PARAM_000+UH10"."I456.2",
             XS_Command := "HMI_CMD_000+UH10"."I456.2",
             OB1Out => "STATUS_000+UH10"."I456.2",
             ENO => #_w2);
   IF #_w2 THEN
       #KF14_Ix3(IB1In := "I456.3",   // "STD_CH_DI"
                 IB1Inv := "STDLog0",
                 XS_Parameter := "HMI_PARAM_000+UH10"."I456.3",
                 XS_Command := "HMI_CMD_000+UH10"."I456.3",
                 OB1Out => "STATUS_000+UH10"."I456.3");
   END_IF;
   #KF14_Ix4(IB1In := "I456.4",   // "STD_CH_DI"
             IB1Inv := "STDLog0",
             XS_Parameter := "HMI_PARAM_000+UH10"."I456.4",
             XS_Command := "HMI_CMD_000+UH10"."I456.4",
             OB1Out => "STATUS_000+UH10"."I456.4",
             ENO => #_w3);
   IF #_w3 THEN
       #KF14_Ix5(IB1In := "I456.5",   // "STD_CH_DI"
                 IB1Inv := "STDLog0",
                 XS_Parameter := "HMI_PARAM_000+UH10"."I456.5",
                 XS_Command := "HMI_CMD_000+UH10"."I456.5",
                 OB1Out => "STATUS_000+UH10"."I456.5");
   END_IF;
   #KF14_Ix6(IB1In := "I456.6",   // "STD_CH_DI"
             IB1Inv := "STDLog0",
             XS_Parameter := "HMI_PARAM_000+UH10"."I456.6",
             XS_Command := "HMI_CMD_000+UH10"."I456.6",
             OB1Out => "STATUS_000+UH10"."I456.6",
             ENO => #_w4);
   IF #_w4 THEN
       #KF14_Ix7(IB1In := "I456.7",   // "STD_CH_DI"
                 IB1Inv := "STDLog0",
                 XS_Parameter := "HMI_PARAM_000+UH10"."I456.7",
                 XS_Command := "HMI_CMD_000+UH10"."I456.7",
                 OB1Out => "STATUS_000+UH10"."I456.7");
   END_IF;
END_REGION
END_FUNCTION_BLOCK
